FUNCTION_BLOCK FB_savePositions
VAR_INPUT
	inputBaseAngle : INT;			// Input baseAngle to be saved to array
	inpitShoulderAngle : INT;		// Input shoulderAngle to be saved to array
	inputElbowAngle : INT;			// Input elbowAngle to be saved to array
	desiredPosIndex : INT;		// Index used to select saved output angles
	isTargetPosReached : BOOL;	// Will increment desiredPosIndex when true
END_VAR
VAR_OUTPUT
	targetBaseAngle : INT;		// baseAngle to be written to servo
	targetShoulderAngle : INT;	// shoulderAngle to be written to servo
	targetElbowAngle : INT;		// elbowAngle to be written to servo
	savedPosCount : INT;		// Number of recorden joint positions
END_VAR
VAR
	currentIndex : INT;			// Index reflecting current saved angles to be written to servos
	savedBasePositions : ARRAY OF INT [0..9] := {-1, -1, -1, -1, -1, -1, -1, -1, -1, -1};		// Saved base positions to be accessed by desiredPosIndex
	savedShoulderPositions : ARRAY OF INT [0..9] := {-1, -1, -1, -1, -1, -1, -1, -1, -1, -1};	// Saved shoulder positions to be accessed by desiredPosIndex
	savedElbowPositions  ARRAY OF INT [0..9] := {-1, -1, -1, -1, -1, -1, -1, -1, -1, -1};		// Saved elbow positions to be accessed by desiredPosIndex
END_VAR

END_FUNCTION_BLOCK

(* stored: Version 1.1.0.1, ProductVersion 3.1.4024.13
   POU FB_savePositions: Id {3f9c5992-6c21-4d73-a6df-987da302f836}, SpecialFunc None *)
